// TIA Portal V19 export
ORGANIZATION_BLOCK "Main"   // OB1, LAD, ProgramCycle
TITLE = "Main Program Sweep (Cycle)"
{ S7_Optimized_Access := 'TRUE' }
AUTHOR : Siemens
// "Main Program
// stored: IsIECCheckEnabled true, SetENOAutomatically true
   VAR_INPUT
      Initial_Call : Bool;   // Initial call of this OB
      Remanence : Bool;   // =True, if remanent data are available
   END_VAR
BEGIN

REGION Network 1
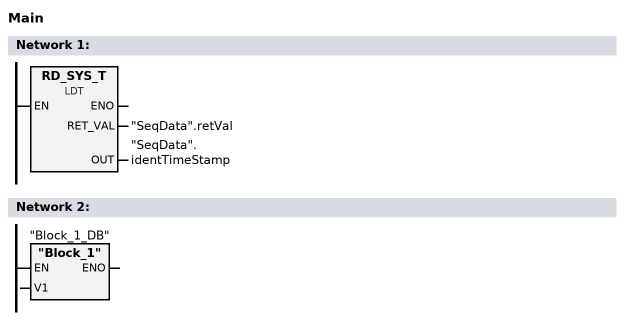
   RUNG wire#powerrail
      { S7_Templates := "date_type := LDT" } RD_SYS_T(RET_VAL => "SeqData".retVal, OUT => "SeqData".identTimeStamp)
   END_RUNG
   // the same network as SCL:
   "SeqData".retVal := RD_SYS_T(OUT => "SeqData".identTimeStamp);
END_REGION

REGION Network 2
   RUNG wire#powerrail
      "Block_1_DB"(V1 :=)
   END_RUNG
   // the same network as SCL:
   "Block_1_DB"();   // "Block_1"
END_REGION
END_ORGANIZATION_BLOCK
